move 81,-240,1.9,0.8,7.7,-8.5;
move 82,-240.2,1.9,0.8,7.8,-8.4;
move 84,-240.5,1.9,1.2,7.9,-8.4;
move 85,-240.8,1.8,1.2,8.1,-8.4;
move 86,-241.1,1.8,1.6,8.2,-8.3;
move 87,-241.5,1.8,1.6,8.3,-8.3;
move 89,-241.8,1.8,2,8.4,-8.2;
move 90,-242.2,1.8,2,8.5,-8.2;
move 91,-242.6,1.8,2,8.6,-8.1;
move 92,-243,1.7,2.4,8.7,-8.1;
move 93,-243.4,1.7,2.4,8.8,-8;
move 94,-243.8,1.7,2.4,8.9,-8;
move 95,-244.1,1.7,2.8,9,-7.9;
move 96,-244.5,1.7,2.8,9.1,-7.9;
move 97,-244.9,1.7,2.8,9.2,-7.8;
move 98,-245.2,1.7,3.2,9.3,-7.8;
move 99,-245.6,1.7,3.2,9.4,-7.7;
move 100,-245.9,1.7,3.6,9.5,-7.7;
move 102,-246.3,1.6,3.6,9.6,-7.6;
move 103,-246.6,1.6,3.6,9.7,-7.6;
move 104,-247,1.6,4,9.8,-7.5;
move 105,-247.3,1.6,4,9.9,-7.5;
move 106,-247.7,1.6,4,10,-7.4;
move 107,-248.1,1.6,4.4,10,-7.4;
move 108,-248.4,1.6,4.4,10.1,-7.3;
move 109,-248.9,1.6,4.4,10.2,-7.3;
move 110,-249.3,1.6,4.8,10.3,-7.2;
move 111,-249.7,1.6,4.8,10.4,-7.1;
move 112,-250.2,1.7,4.8,10.5,-7.1;
move 113,-250.7,1.7,5.2,10.6,-7;
move 114,-251.2,1.7,5.2,10.7,-7;
move 115,-251.7,1.7,5.2,10.8,-6.9;
move 116,-252.3,1.7,5.6,10.9,-6.8;
move 117,-252.8,1.7,5.6,10.9,-6.8;
move 118,-253.4,1.7,6,11,-6.7;
move 119,-254,1.7,6,11.1,-6.7;
move 120,-254.6,1.7,6,11.2,-6.6;
move 121,-255.2,1.7,6.4,11.3,-6.5;
move 122,-255.8,1.7,6.4,11.4,-6.5;
move 123,-256.5,1.7,6.4,11.4,-6.4;
move 124,-257.1,1.7,6.4,11.5,-6.3;
move 125,-257.7,1.7,6.8,11.6,-6.3;
move 125,-258.3,1.7,6.8,11.7,-6.2;
move 126,-258.9,1.8,6.8,11.8,-6.2;
move 127,-259.5,1.8,7.2,11.8,-6.1;
move 128,-260.1,1.8,7.2,11.9,-6;
move 129,-260.6,1.8,7.2,12,-6;
move 130,-261.1,1.8,7.6,12.1,-5.9;
move 131,-261.6,1.8,7.6,12.1,-5.8;
move 132,-262.1,1.8,7.6,12.2,-5.8;
move 133,-262.6,1.8,8,12.3,-5.7;
move 134,-263.1,1.8,8,12.3,-5.6;
move 135,-263.5,1.8,8,12.4,-5.5;
move 137,-264,1.8,8.4,12.5,-5.5;
move 138,-264.4,1.8,8.4,12.6,-5.4;
move 139,-264.8,1.8,8.8,12.6,-5.3;
move 140,-265.2,1.8,8.8,12.7,-5.3;
move 141,-265.6,1.8,8.8,12.8,-5.2;
move 142,-266,1.8,9.2,12.8,-5.1;
move 143,-266.4,1.8,9.2,12.9,-5.1;
move 144,-266.9,1.8,9.2,13,-5;
move 146,-267.3,1.8,9.6,13,-4.9;
move 147,-267.8,1.8,9.6,13.1,-4.8;
move 148,-268.3,1.8,10,13.1,-4.8;
move 149,-268.8,1.8,10,13.2,-4.7;
move 151,-269.4,1.8,10.4,13.3,-4.6;
move 152,-270,1.8,10.4,13.3,-4.5;
move 153,-270.7,1.7,10.4,13.4,-4.5;
move 154,-271.4,1.7,10.8,13.4,-4.4;
move 156,-272.1,1.7,10.8,13.5,-4.3;
move 157,-272.9,1.7,11.2,13.5,-4.3;
move 158,-273.7,1.7,11.2,13.6,-4.2;
move 159,-274.6,1.7,11.6,13.6,-4.1;
move 161,-275.5,1.7,11.6,13.7,-4;
move 162,-276.4,1.6,11.6,13.7,-4;
move 163,-277.4,1.6,12,13.8,-3.9;
move 164,-278.4,1.6,12,13.8,-3.8;
move 166,-279.4,1.6,12.4,13.9,-3.8;
move 167,-280.5,1.6,12.4,13.9,-3.7;
move 168,-281.6,1.5,12.8,14,-3.6;
move 169,-282.8,1.5,12.8,14,-3.6;
move 171,-283.9,1.5,12.8,14.1,-3.5;
move 172,-285.1,1.5,13.2,14.1,-3.5;
move 173,-286.3,1.5,13.2,14.2,-3.4;
move 175,-287.4,1.4,13.6,14.2,-3.3;
move 176,-288.6,1.4,13.6,14.2,-3.3;
move 178,-289.7,1.4,14,14.3,-3.2;
move 179,-290.9,1.3,14,14.3,-3.2;
move 180,-292,1.3,14.4,14.4,-3.1;
move 182,-293.1,1.3,14.4,14.4,-3;
move 183,-294.3,1.2,14.8,14.4,-3;
move 185,-295.4,1.2,14.8,14.5,-2.9;
move 186,-296.4,1.2,15.2,0,-2.9;
move 188,-297.5,1.1,15.2,0,-2.8;
move 189,-298.5,1.1,15.6,0,-2.8;
move 191,-299.6,1.1,15.6,0,-2.7;
move 192,-300.5,1,16,0,-2.7;
move 194,-301.5,1,16,0,-2.7;
move 195,-302.4,1,16.4,0,-2.6;
move 196,-303.3,0.9,16.4,0,-2.6;
move 198,-304.1,0.9,16.8,0,-2.5;
move 199,-304.9,0.9,16.8,0,-2.5;
move 200,-305.7,0.8,17.2,0,-2.5;
move 201,-306.5,0.8,17.2,0,-2.4;
move 202,-307.2,0.7,17.6,0,-2.4;
move 203,-307.9,0.7,17.6,0,-2.4;
move 203,-308.6,0.7,17.6,0,-2.3;
move 204,-309.2,0.6,18,0,-2.3;




    ENDPROC

! function used to produce movement
    PROC move(num x, num z,num rx, num ry, num rz,num joint1)
     ConfJ\On;
     velocity := [300,1000,5000,1000];

     !IF (ry<(10) AND ry>(-10)) THEN
     !   velocity := v300;
     !ELSE
     !   velocity:=v600;
     !ENDIF


     !!!! Method Two !!!!!!
     position :=RelTool(starting_position, x,0, z \Rx:=rx, \Ry:=ry, \Rz:=rz);
     joints := CalcJointT(position,Tooldata_9 \WObj:=Workobject_2);
     joints.robax.rax_1 :=joint1;
     MoveAbsJ joints,velocity,z200,Tooldata_9,\WObj:=wobj0;
     !!!!!!!!!!!!!!!!!!!!!!!!!!!!!!
   ! MoveJ RelTool (starting_position, x,0, z \Rx:=rx, \Ry:=ry, \Rz:=0),v200,fine,Tooldata_9 \WObj:=Workobject_2;
   ! joints := CJointT(\TaskName:="T_ROB1");
   ! joints.robax.rax_1 := joint1;
    !MoveAbsJ joints,v200,fine,tool0,\WObj:=wobj0;
    !!!!!!!!!!!!!!!!!!!!!!!!!!!!!!!!!!!!!!!
    ENDPROC



ENDMODULE
